(* CoDeSys 2.3.9.28 project: Aula10_CAFES_FINAL.pro *)
(* Libraries: Standard.lib 4.10.05 12:14:46, Util.lib 18.5.10 15:14:28, IecSfc.lib 13.4.06 15:51:28, SysLibTime.lib 27.1.09 11:27:38, SysTaskInfo.lib 24.11.08 08:07:15, SYSLIBCALLBACK.LIB 27.1.09 11:27:38 *)

(* Global variable list: Global_Variables *)
VAR_GLOBAL

	B1 : BOOL;
	B2 : BOOL;
	B3 : BOOL;

	A1 : BOOL;
	A2 : BOOL;
	A3 : BOOL;

	SC : BOOL;
	BP : BOOL;
	OK : BOOL;


	VR1 AT %QX0.0 : BOOL;
	VR2 AT %QX0.1 : BOOL;
	VR3 AT %QX0.2 : BOOL;
	VR4 AT %QX0.3 : BOOL;
	VR5 AT %QX0.4 : BOOL;
	AC AT %QX0.5 : BOOL;
	LP AT %QX0.6 : BOOL;

	T1 : TOF;
	T2 : TOF;
	T3 : TOF;
	T4_2 : TON;
	T4_3 : TON;
	T5 : TOF;
	T_AGUA : TON;

	MEM : BOOL;
	MEM1 : BOOL;
	MEM3 : BOOL;
	MEM_PA : BOOL;
	MEM_MA : BOOL;

	MEM_SABOR : BOOL;
	MEM_ACUCAR : BOOL;

	MEM_A1 : BOOL;
	MEM_A2 : BOOL;
	MEM_A3 : BOOL;
	MEM_B1 : BOOL;
	MEM_B2 : BOOL;
	MEM_B3 : BOOL;


	CONT1 : CTU;



END_VAR

(* POU PLC_PRG, LD *)
PROGRAM PLC_PRG
VAR

END_VAR
VAR (* helpers for the ST form of the networks *)
	_p1 : BOOL;
	_p2 : BOOL;
	_p3 : BOOL;
	_p4 : BOOL;
	_p5 : BOOL;
	_p6 : BOOL;
	_p7 : BOOL;
END_VAR
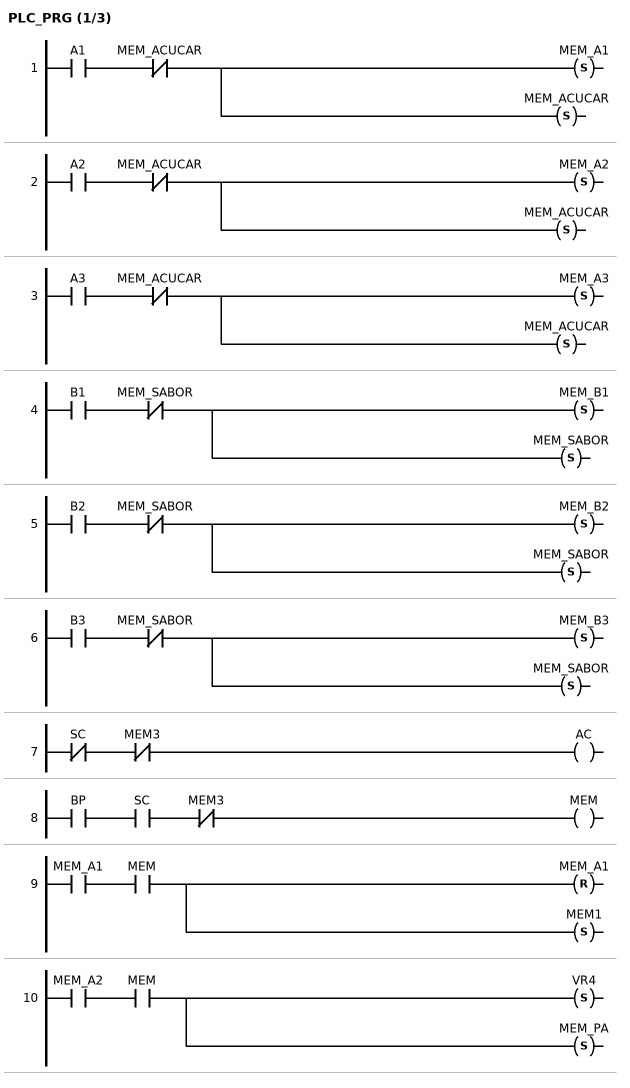
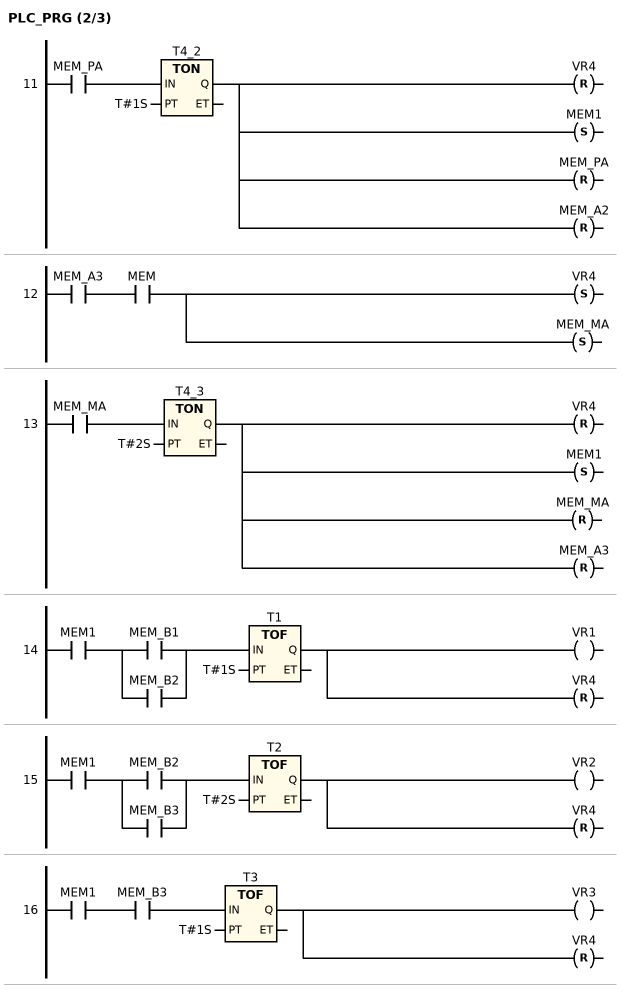
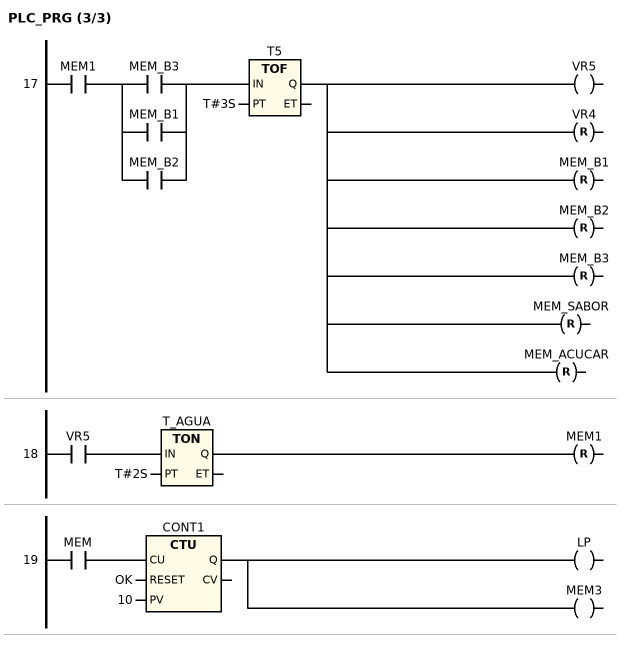
_LD_ (* Ladder Diagram *)
NETWORK 1
	[A1] - [/MEM_ACUCAR] --- (S MEM_A1) (S MEM_ACUCAR)
NETWORK 2
	[A2] - [/MEM_ACUCAR] --- (S MEM_A2) (S MEM_ACUCAR)
NETWORK 3
	[A3] - [/MEM_ACUCAR] --- (S MEM_A3) (S MEM_ACUCAR)
NETWORK 4
	[B1] - [/MEM_SABOR] --- (S MEM_B1) (S MEM_SABOR)
NETWORK 5
	[B2] - [/MEM_SABOR] --- (S MEM_B2) (S MEM_SABOR)
NETWORK 6
	[B3] - [/MEM_SABOR] --- (S MEM_B3) (S MEM_SABOR)
NETWORK 7
	[/SC] - [/MEM3] --- (AC)
NETWORK 8
	[BP] - [SC] - [/MEM3] --- (MEM)
NETWORK 9
	[MEM_A1] - [MEM] --- (R MEM_A1) (S MEM1)
NETWORK 10
	[MEM_A2] - [MEM] --- (S VR4) (S MEM_PA)
NETWORK 11
	[MEM_PA] - T4_2:TON(IN: *, PT: T#1S) --- (R VR4) (S MEM1) (R MEM_PA) (R MEM_A2)
NETWORK 12
	[MEM_A3] - [MEM] --- (S VR4) (S MEM_MA)
NETWORK 13
	[MEM_MA] - T4_3:TON(IN: *, PT: T#2S) --- (R VR4) (S MEM1) (R MEM_MA) (R MEM_A3)
NETWORK 14
	[MEM1] - { [MEM_B1] | [MEM_B2] } - T1:TOF(IN: *, PT: T#1S) --- (VR1) (R VR4)
NETWORK 15
	[MEM1] - { [MEM_B2] | [MEM_B3] } - T2:TOF(IN: *, PT: T#2S) --- (VR2) (R VR4)
NETWORK 16
	[MEM1] - [MEM_B3] - T3:TOF(IN: *, PT: T#1S) --- (VR3) (R VR4)
NETWORK 17
	[MEM1] - { [MEM_B3] | [MEM_B1] | [MEM_B2] } - T5:TOF(IN: *, PT: T#3S) --- (VR5) (R VR4) (R MEM_B1) (R MEM_B2) (R MEM_B3) (R MEM_SABOR) (R MEM_ACUCAR)
NETWORK 18
	[VR5] - T_AGUA:TON(IN: *, PT: T#2S) --- (R MEM1)
NETWORK 19
	[MEM] - CONT1:CTU(CU: *, RESET: OK, PV: 10) --- (LP) (MEM3)
_END_LD_
(* the same logic as Structured Text *)
(* Network 1 *)
_p1 := A1 AND NOT MEM_ACUCAR;
IF _p1 THEN MEM_A1 := TRUE; MEM_ACUCAR := TRUE; END_IF;
(* Network 2 *)
_p2 := A2 AND NOT MEM_ACUCAR;
IF _p2 THEN MEM_A2 := TRUE; MEM_ACUCAR := TRUE; END_IF;
(* Network 3 *)
_p3 := A3 AND NOT MEM_ACUCAR;
IF _p3 THEN MEM_A3 := TRUE; MEM_ACUCAR := TRUE; END_IF;
(* Network 4 *)
_p4 := B1 AND NOT MEM_SABOR;
IF _p4 THEN MEM_B1 := TRUE; MEM_SABOR := TRUE; END_IF;
(* Network 5 *)
_p5 := B2 AND NOT MEM_SABOR;
IF _p5 THEN MEM_B2 := TRUE; MEM_SABOR := TRUE; END_IF;
(* Network 6 *)
_p6 := B3 AND NOT MEM_SABOR;
IF _p6 THEN MEM_B3 := TRUE; MEM_SABOR := TRUE; END_IF;
(* Network 7 *)
AC := NOT SC AND NOT MEM3;
(* Network 8 *)
MEM := BP AND SC AND NOT MEM3;
(* Network 9 *)
_p7 := MEM_A1 AND MEM;
IF _p7 THEN MEM_A1 := FALSE; MEM1 := TRUE; END_IF;
(* Network 10 *)
IF MEM_A2 AND MEM THEN VR4 := TRUE; MEM_PA := TRUE; END_IF;
(* Network 11 *)
T4_2(IN := MEM_PA, PT := T#1S);
IF T4_2.Q THEN VR4 := FALSE; MEM1 := TRUE; MEM_PA := FALSE; MEM_A2 := FALSE; END_IF;
(* Network 12 *)
IF MEM_A3 AND MEM THEN VR4 := TRUE; MEM_MA := TRUE; END_IF;
(* Network 13 *)
T4_3(IN := MEM_MA, PT := T#2S);
IF T4_3.Q THEN VR4 := FALSE; MEM1 := TRUE; MEM_MA := FALSE; MEM_A3 := FALSE; END_IF;
(* Network 14 *)
T1(IN := MEM1 AND (MEM_B1 OR MEM_B2), PT := T#1S);
VR1 := T1.Q;
IF T1.Q THEN VR4 := FALSE; END_IF;
(* Network 15 *)
T2(IN := MEM1 AND (MEM_B2 OR MEM_B3), PT := T#2S);
VR2 := T2.Q;
IF T2.Q THEN VR4 := FALSE; END_IF;
(* Network 16 *)
T3(IN := MEM1 AND MEM_B3, PT := T#1S);
VR3 := T3.Q;
IF T3.Q THEN VR4 := FALSE; END_IF;
(* Network 17 *)
T5(IN := MEM1 AND (MEM_B3 OR MEM_B1 OR MEM_B2), PT := T#3S);
VR5 := T5.Q;
IF T5.Q THEN VR4 := FALSE; END_IF;
IF T5.Q THEN MEM_B1 := FALSE; END_IF;
IF T5.Q THEN MEM_B2 := FALSE; END_IF;
IF T5.Q THEN MEM_B3 := FALSE; END_IF;
IF T5.Q THEN MEM_SABOR := FALSE; END_IF;
IF T5.Q THEN MEM_ACUCAR := FALSE; END_IF;
(* Network 18 *)
T_AGUA(IN := VR5, PT := T#2S);
IF T_AGUA.Q THEN MEM1 := FALSE; END_IF;
(* Network 19 *)
CONT1(CU := MEM, RESET := OK, PV := 10);
LP := CONT1.Q;
MEM3 := CONT1.Q;
END_PROGRAM

(* Visualisation View01
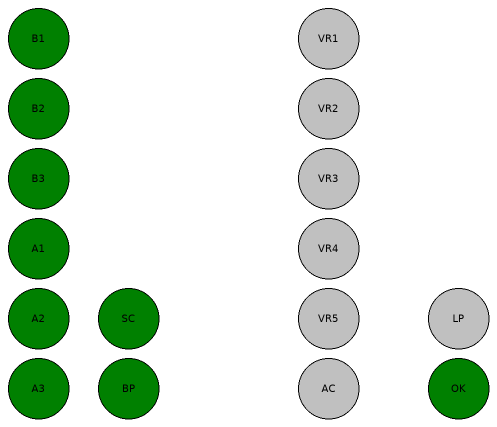
ellipse at (30,20)-(91,81): text "B1"; alarm colour if B1; taps B1
ellipse at (450,300)-(511,361): text "LP"; alarm colour if LP
ellipse at (30,90)-(91,151): text "B2"; alarm colour if B2; taps B2
ellipse at (30,160)-(91,221): text "B3"; alarm colour if B3; taps B3
ellipse at (30,230)-(91,291): text "A1"; alarm colour if A1; taps A1
ellipse at (30,300)-(91,361): text "A2"; alarm colour if A2; taps A2
ellipse at (30,370)-(91,431): text "A3"; alarm colour if A3; taps A3
ellipse at (320,370)-(381,431): text "AC"; alarm colour if AC
ellipse at (320,20)-(381,81): text "VR1"; alarm colour if VR1
ellipse at (320,90)-(381,151): text "VR2"; alarm colour if VR2
ellipse at (320,160)-(381,221): text "VR3"; alarm colour if VR3
ellipse at (320,230)-(381,291): text "VR4"; alarm colour if VR4
ellipse at (320,300)-(381,361): text "VR5"; alarm colour if VR5
ellipse at (120,300)-(181,361): text "SC"; alarm colour if SC; toggles SC
ellipse at (120,370)-(181,431): text "BP"; alarm colour if BP; taps BP
ellipse at (450,370)-(511,431): text "OK"; alarm colour if OK; taps OK
*)
